TYPE ParametersPosition :
STRUCT
	Velocity : LREAL := 50; //in mm/s
	Acceleration: LREAL := 500; // in mm/s2
	Deceleration: LREAL := 500;
	Position: LREAL := 10; // in mm
END_STRUCT
END_TYPE

(* stored: Version 1.1.0.1, ProductVersion 3.1.4022.10
   DUT ParametersPosition: Id {85e9894d-ac1a-4d9d-9bd7-9be3113bbb94} *)
